FUNCTION F_LeakBoundaries : ST_LeakBoundaries
VAR_INPUT
END_VAR
VAR
	stLeakBoundaries : ST_LeakBoundaries := (
		nLMin1 := 0,
		nLMax1 := 1000,
		nLMin2 := 1000,
		nLMax2 := 2000,
		nLMin3 := 2000,
		nLMax3 := 3000,
		nLMin4 := 3000,
		nLMax4 := 4000,
		nLMin5 := 4000,
		nLMax5 := 5000,
		nLMin6 := 5000,
		nLMax6 := 6000
	);
END_VAR

F_LeakBoundaries := stLeakBoundaries;

END_FUNCTION

(* stored: Version 1.1.0.1, ProductVersion 3.1.4020.14
   POU F_LeakBoundaries: Id {d9d75f4b-af19-479d-9bc9-5809cb8f372a}, SpecialFunc None *)
